(* Schneider Machine Expert - Basic project demo1_config, file version 2.2.0.0 *)
(* CompanyInformations: WebSite=https://ics-cybersecurity.com *)
(* ProjectInformations: Name=ICSJWG example 1, Description=Very simple example to enable/disable some of the communication protocols *)
(* UserInformations: LastName=Arnaud, FirstName=SOULLIE, Email=asoullie@ics-cybersecurity.academy *)

HARDWARE
  Cpu 0: TM221ME16R/G
  EthernetConfiguration: NetworkName=M221, IpAllocationMode=FixedAddress, IpAddress=192.168.0.53, SubnetMask=255.255.255.0
  SerialLineConfiguration: Baud=Baud19200, Parity=ParityEven, DataBits=DataBits8, StopBits=StopBits1, PhysicalMedium=PhysicalMediumRs485, TransmissionMode=TransmissionModeModbusRtu, SlaveId=1, Addressing=SlaveAddressing
  MastTask: UsePeriodScanMode=false, PeriodScan=100
  FastTask: Period=255
  CpuBehavior: StartingMode=StartAsPreviousState, AutoSaveRamOnEeprom=true, WatchdogPeriod=250

SYMBOLS  (address, symbol, comment, settings)
  %M0       HEATING_START
  %M20      WASH_INTAKE
  %M23      BARREL_VALVE
  %M100     IO_FORCED
  %M101     INPUT_FORCED
  %M102     OUTPUT_FORCED
  %MW0      HEATING_DURATION
  %MW10     STILL_TEMP
  %MW11     STILL_LEVEL
  %MW12     CONDENSER_TEMP
  %MW13     BARREL_LEVEL
  %MW21     HEATER
  %MW22     COOLING_PUMP
  %MW100    BOOTLOADER_VERSION
  %MW101    COMMERCIAL_VERSION
  %MW102    FIRMWARE_V_PART1
  %MW103    FIRMWARE_V_PART2
  %MW104    APPLICATION_SIGNATURE
  %MW110    LAST_SCAN_TIME

POU New POU
  (* SectionNumber=1 *)

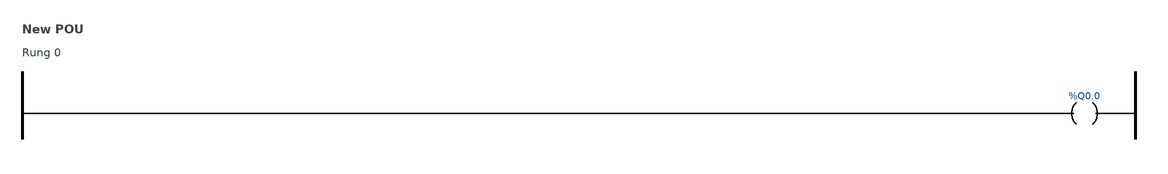

// Rung 0
  LD 1
  ST %Q0.0
  // as ST:
  //   %Q0.0 := TRUE;
